FUNCTION_BLOCK FB_Zylinder
VAR_INPUT
	bGate : BOOL;
	bError : BOOL;
END_VAR

VAR_OUTPUT
	bR1 : BOOL;
	bR2 : BOOL;
END_VAR

VAR
END_VAR

bR1 := bGate;
bR2 := NOT bGate;

IF bError THEN
	br1 := FALSE;
	br2 := FALSE;
END_IF

END_FUNCTION_BLOCK

(* stored: Version 1.1.0.1, ProductVersion 3.1.4024.15
   POU FB_Zylinder: Id {2fed519a-143f-4e3d-b67a-c4f039b2c945}, SpecialFunc None *)
